FUNCTION_BLOCK FB_Blinker
VAR_INPUT
	TmrPreset : TIME;
END_VAR
VAR_OUTPUT
	xOut : BOOL;
END_VAR
VAR
	xBlink : BOOL;	
	xBlinkOFF : BOOL;	
	BlinkTmr : TON;
	BlinkOffTmr : TON;
	BlinkDly : TON;
END_VAR

BlinkDly(IN:= TRUE, PT:= T#1S , Q=> , ET=> );

IF BlinkDly.Q THEN
	BlinkTmr(IN:= NOT xBlinkOFF , PT:= TmrPreset, Q=> xBlink , ET=> );
	BlinkOFFTmr(IN:= xBlink, PT:= TmrPreset, Q=> xBlinkOFF , ET=> );
	xOut := xBlink;
ELSE
	xBlink := FALSE;
END_IF

END_FUNCTION_BLOCK

(* stored: Version 1.1.0.1, ProductVersion 3.1.4024.14
   POU FB_Blinker: Id {5d5c7b60-d19f-4dd0-9617-1f387e579ef8}, SpecialFunc None *)
